// TwinCAT 3 PLC project Untitled1
// ProgramVersion: 3.1.4023.0
// libraries:
//   Tc2_EthernetIP, * (Beckhoff Automation GmbH)
//   Tc2_MC2, * (Beckhoff Automation GmbH)
//   Tc2_Standard, * (Beckhoff Automation GmbH)
//   Tc2_System, * (Beckhoff Automation GmbH)
//   Tc2_TcpIp, * (Beckhoff Automation GmbH)
//   Tc2_Utilities, * (Beckhoff Automation GmbH)
//   Tc3_Interfaces, * (Beckhoff Automation GmbH)
//   Tc3_Module, * (Beckhoff Automation GmbH)
//   VisuDialogs, * (System)
// project tree:
//   DUTs/ ST_Handshake.TcDUT, ST_Input_Output.TcDUT
//   / GlobalTextList.TcGTLO, PlcTask.TcTTO, Visualization Manager.TcVMO (not stored)
//   GVLs/ Global_Variables.TcGVL, GVL.TcGVL
//   POUs/ FB_Server.TcPOU, FB_ServerApplication.TcPOU, FB_ServerConnection.TcPOU, MAIN.TcPOU, Torque.TcPOU, Velocity.TcPOU
//   POUs/Helper POUs/ FB_FrameFifo.TcPOU, FB_LogFifo.TcPOU, F_ADSLOGHEXDATA.TcPOU
//   VISUs/ Visualization.TcVIS
// real-time tasks:
//   TASK PlcTask: cycle T#100us, priority 20, ADS port 350
// motion (NC):
//   TASK NC-Task 1 SAF: cycle T#2ms, priority 4, ADS port 501
//   TASK NC-Task 1 SVB: cycle T#10ms, priority 8, ADS port 511
//   AXIS Axis 1 (id 1)
//     OtherSettings: AllowMotionCmdToSlave=true
//     encoder EncType=4
//       EncPara: MaxCount=#x0000ffff
//         Inc: RefSoftSyncMask=#x0000ffff
//     drive DrvType=24
//       Analog: TorqueSetpointScale=10, ScaleFactorActTorque=0.1
//       TimeComp: TaskDelayCycles=1
//     controller CtrType=1
//       CtrPara: PriorControlFactor=1
//         Observer: BandWidth=20
//   AXIS Axis 2 (id 2)
//     Dynamic: Acceleration=193.102849139388, Deceleration=193.102849139388, Jerk=13.317479191567
//     Velo: RefSearch=28.7326666666667, RefSync=28.7326666666667, SlowManual=143.663333333333, FastManual=861.98, Fast=2873.26666666667, Maximum=2800
//     PositionAreaControl: Enable=false
//     TargetPosControl: Enable=false
//     OtherSettings: AllowMotionCmdToSlave=true
//     encoder EncType=19
//       EncPara: ScaleFactorNumerator=94, ScaleFactorDenominator=1048576, MaxCount=#xffffffff
//     drive DrvType=16
//       DrvPara: MaxCount=#xffffffff
//         Analog: VeloReferenz=3000, VeloScale=32, TorqueSetpointScale=10, ScaleFactorActTorque=0.1
//         TimeComp: TaskDelayCycles=1
//     controller CtrType=1
//       CtrPara: PriorControlFactor=1
//         PosDiffControl: Enable=false
//         Observer: BandWidth=20
//   AXIS Axis 3 (id 3)
//     OtherSettings: AllowMotionCmdToSlave=true
//     encoder EncType=19
//       EncPara: ScaleFactorNumerator=104.8576, ScaleFactorDenominator=1048576, MaxCount=#xffffffff
//     drive DrvType=16
//       DrvPara: MaxCount=#xffffffff, DriveControlDWord=#x00020000
//         Analog: VeloScale=32, TorqueSetpointScale=10, ScaleFactorActTorque=0.1
//         TimeComp: TaskDelayCycles=1
//     controller CtrType=1
//       CtrPara: PriorControlFactor=1
//         Observer: BandWidth=20
// I/O:
//   DEVICE Device 1 (EtherCAT), AmsNetId 192.168.0.4.2.1
//     Term 13 (EK1200) [EK1200-5000 EtherCAT Power supply (2A E-Bus)]
//       Term 14 (EL1004) [EL1004 4Ch. Dig. Input 24V, 3ms]
//       Term 15 (EL1008) [EL1008 8Ch. Dig. Input 24V, 3ms]
//       Term 16 (EL2004) [EL2004 4Ch. Dig. Output 24V, 0.5A]
//       Term 17 (EL2008) [EL2008 8Ch. Dig. Output 24V, 0.5A]
//       Term 18 (EL3102) [EL3102 2Ch. Ana. Input +/-10V, Diff.]
//       Term 19 (EL4132) [EL4132 2Ch. Ana. Output +/-10V, 16bit]
//       Term 20 (EK1110) [EK1110 EtherCAT extension]
//     Term 21 (EK1100) [EK1100 EtherCAT Coupler (2A E-Bus)]
//       Term 22 (EL7031) [EL7031 1Ch. Stepper motor output stage (24V, 1.5A)]
//       Term 23 (EL7211-0010) [EL7211-0010 1Ch. MDP742 Servo motor output stage with OCT (50V, 4.5A RMS)]
//       Term 27 (EL9011) [EL9011 End Terminal]
//     Term 24 (EK1100) [EK1100 EtherCAT Coupler (2A E-Bus)]
//       Term 25 (EL7211-0010) [EL7211-0010 1Ch. MDP742 Servo motor output stage with OCT (50V, 4.5A RMS)]
//       Term 26 (EK1110) [EK1110 EtherCAT extension]
//   DEVICE Device 5 (COM Port)
// variable links:
//   NC-Task 1 SAF/Axes/Axis 2 <-> Device 1 (EtherCAT)/Term 21 (EK1100)/Term 23 (EL7211-0010)
//     Drive/Inputs/In/nDataIn3[0] <-> DRV Torque actual value/Torque actual value
//     Drive/Inputs/In/nDcOutputTime <-> InfoData/DcOutputShift
//     Drive/Inputs/In/nState1 <-> DRV Statusword/Statusword
//     Drive/Inputs/In/nState2 <-> DRV Statusword/Statusword @bit 8
//     Drive/Inputs/In/nState4 @bit 1 <-> WcState/InputToggle
//     Drive/Inputs/In/nState4 <-> WcState/WcState
//     Drive/Outputs/Out/nCtrl1 <-> DRV Controlword/Controlword
//     Drive/Outputs/Out/nCtrl2 <-> DRV Controlword/Controlword @bit 8
//     Enc/Inputs/In/nDataIn1 <-> FB Position/Position
//     Enc/Inputs/In/nDcInputTime <-> InfoData/DcInputShift
//     Enc/Inputs/In/nState4 @bit 1 <-> WcState/InputToggle
//     Enc/Inputs/In/nState4 <-> WcState/WcState
//   NC-Task 1 SAF/Axes/Axis 3 <-> Device 1 (EtherCAT)/Term 24 (EK1100)/Term 25 (EL7211-0010)
//     Drive/Inputs/In/nDcOutputTime <-> InfoData/DcOutputShift
//     Drive/Inputs/In/nState1 <-> DRV Statusword/Statusword
//     Drive/Inputs/In/nState2 <-> DRV Statusword/Statusword @bit 8
//     Drive/Inputs/In/nState4 @bit 1 <-> WcState/InputToggle
//     Drive/Inputs/In/nState4 <-> WcState/WcState
//     Drive/Outputs/Out/nCtrl1 <-> DRV Controlword/Controlword
//     Drive/Outputs/Out/nCtrl2 <-> DRV Controlword/Controlword @bit 8
//     Drive/Outputs/Out/nDataOut2 <-> DRV Target velocity/Target velocity
//     Enc/Inputs/In/nDataIn1 <-> FB Position/Position
//     Enc/Inputs/In/nDcInputTime <-> InfoData/DcInputShift
//     Enc/Inputs/In/nState4 @bit 1 <-> WcState/InputToggle
//     Enc/Inputs/In/nState4 <-> WcState/WcState
//   Untitled1/Untitled1 Instance <-> Device 1 (EtherCAT)/Term 21 (EK1100)/Term 23 (EL7211-0010)
//     PlcTask Outputs/Torque.TorqueLim <-> DRV Torque limitation/Torque limitation
//     PlcTask Outputs/Torque.TorqueVAL <-> DRV Target torque/Target torque
//   Untitled1/Untitled1 Instance <-> NC-Task 1 SAF/Axes/Axis 2
//     PlcTask Inputs/GVL.ActualTorque <-> Outputs/ToPlc/ActTorque
//     PlcTask Inputs/Torque.Axis1.NcToPlc <-> Outputs/ToPlc
//     PlcTask Outputs/Torque.Axis1.PlcToNc <-> Inputs/FromPlc
//   Untitled1/Untitled1 Instance <-> NC-Task 1 SAF/Axes/Axis 3
//     PlcTask Inputs/Velocity.Axis2.NcToPlc <-> Outputs/ToPlc
//     PlcTask Outputs/Velocity.Axis2.PlcToNc <-> Inputs/FromPlc

CONFIGURATION Untitled1
    RESOURCE PLC ON TwinCAT3
        TASK PlcTask(INTERVAL := T#100us, PRIORITY := 20);
        PROGRAM Torque WITH PlcTask : Torque;
        PROGRAM Velocity WITH PlcTask : Velocity;
        PROGRAM MAIN WITH PlcTask : MAIN;
    END_RESOURCE
END_CONFIGURATION

// ---- DUTs/ST_Handshake.TcDUT
TYPE ST_Handshake :
STRUCT
	(* Handshake with Mevea. First package to sent to Mevea. Mevea sends similar, but in diffrent order after connection. These must match.*)
	
	in			: UDINT		:= 3;(* Input parameter amount. 4 byte *)
	out			: UDINT		:= 3;(* Output parameter amount. 4 byte *)
	version	 	: UDINT		:= 1;(* Version. 4 byte *)

	(* Total user data size = 12 byte *)
END_STRUCT
END_TYPE

// ---- DUTs/ST_Input_Output.TcDUT
TYPE ST_Input_Output :
STRUCT
	(* data struct to be transferred with Mevea. Not ideal, but simple to implement and does the trick in this case *)
	
	brake				: LREAL		:= 0;(* 8 byte *)
	rpmin_torqout	 	: LREAL		:= 0;(* 8 byte *)
	rpmout_speedin		: LREAL		:= 0;(* 8 byte *)

	(* Total user data size = 24 bytes *)
END_STRUCT
END_TYPE

// ---- GVLs/Global_Variables.TcGVL
VAR_GLOBAL CONSTANT
	PLCPRJ_BUFFER_SIZE						: UDINT := 1000;	(* Max. internal fifo/receiver buffer size *)
	PLCPRJ_RECEIVE_POLLING_TIME				: TIME := T#0MS;	(* Input polling timer if needed to limit the interval. Not in this case *)
	PLCPRJ_RECEIVE_TIMEOUT					: TIME := T#10S;	(* Timeout when receiving. Start waiting new connection. Usually disconnected by peer error triggers it *)

	(* Some project specific error codes *)
	PLCPRJ_ERROR_RECEIVE_TIMEOUT			: UDINT := 16#8101;(* Receive timeout *)
	PLCPRJ_ERROR_SENDFIFO_OVERFLOW			: UDINT := 16#8102;(* Send fifo overflow *)
	PLCPRJ_ERROR_RECFIFO_OVERFLOW			: UDINT := 16#8103;(* Receive fifo overflow *)
	PLCPRJ_ERROR_INVALID_FRAME_FORMAT		: UDINT := 16#8104;(* Invalid frame format/data *)
	
	PLCPRJ_CRUISE_CONTROL_SET				: LREAL := 20;	(* Max. internal fifo/receiver buffer size *)
END_VAR

// ---- GVLs/GVL.TcGVL
VAR_GLOBAL
	maxSimulationTorque: INT;
	maxSimulationVelocity: INT;
	Actual_Velocity: LREAL;
	ActualTorque AT %I*: LREAL;
	(* Velocity and torque datatype should be given a thought. If there is no reason for int, LREAL would be more suitable *)
	SetVelocity: INT;
	SetTorque: INT;
END_VAR

// ---- POUs/Torque.TcPOU
PROGRAM Torque
VAR
	res1Error: BOOL;
	Step: INT;
	Axis1_MV: MC_MoveVelocity;
	Axis1_Error_Reset: MC_Reset;
	Power1_BufferMode: MC_BufferMode;
	Power1_Override: LREAL;
	Power1_EnableNeg: BOOL;
	Power1_EnablePos: BOOL;
	Power1_Enable: BOOL;
	Axis1_Power: MC_Power;
	Axis1: AXIS_REF;
	Power1_Status: BOOL;
	Power1_Busy: BOOL;
	Power1_error: BOOL;
	Power1_Active: BOOL;
	Power1_ErrorID: UDINT;
	ErrorReset1_Execute: BOOL;
	res1Done: BOOL;
	res1Busy: BOOL;
	res1ErrorID: UDINT;
	MV1_Execute: BOOL;
	MV1_Done: BOOL;
	MV1_Velocity: LREAL;
	MV1_Decceleration: LREAL;
	MV1_Jerk: LREAL;
	MV1_Direction: MC_Direction;
	MV1_Buffermode: MC_BufferMode;
	MV1_InVelocity: BOOL;
	MV1_Busy: BOOL;
	MV1_CommandAborted: BOOL;
	MV1_Error: BOOL;
	MV1_ErrorID: UDINT;
	MV1_Acceleration: LREAL;
	MV1_Accelleration: LREAL;
	MV1_Active: BOOL;
	TorqueVAL AT %Q*: INT;
	TorqueLim AT %Q*: UINT;
	Start1Btn: BOOL;
	PowerOnTorqueBtn: BOOL;
	Stop1Btn: BOOL;
	TorqueEnable: BOOL;
	
	TorqueSim: INT;
END_VAR

//Torque Controlled Servo
	
	//In case of an error with torque controlled servo:
	IF(Power1_error = TRUE OR MV1_Error=TRUE)THEN
		//Step := 10;
	END_IF
	
	//Enables user to set the torque of the servomotor
	IF TorqueEnable  = TRUE THEN
		TorqueVAL := SetTorque;
		TorqueSim := SetTorque*maxSimulationTorque;
	END_IF
	CASE Step OF
		0://Start of the power (in next step), when the PowerOnTorque button will be clicked
			IF (PowerOnTorqueBtn = TRUE) THEN
				Step := 1;
			END_IF
		1://Start the torque control, when the StartTorque button will be clicked
	Axis1_Power(
	Axis:=Axis1,
	Enable := TRUE,
	Enable_Positive := TRUE,
	Enable_Negative := TRUE,
	Override := 100,
	BufferMode := Power1_BufferMode,
	Status => Power1_Status,
	Busy => Power1_Busy,
	Active => Power1_Active,
	Error => Power1_error,
	ErrorID =>Power1_ErrorID);
			IF (Start1Btn = TRUE) THEN
				Step := 2;
				PowerOnTorqueBtn := FALSE;
			END_IF
		2://Stop the motor (in next step), when the StopTorque button will be clicked 
			TorqueLim := 200;
			TorqueEnable := TRUE;
			Start1Btn := FALSE;
			Axis1_MV(
	Axis:= Axis1, 
	Execute:= TRUE, 
	//Velocity:= MV1_Velocity, 
	//Acceleration:= MV1_Accelleration, 
	//Deceleration:= MV1_Decceleration, 
	//Jerk:= MV1_Jerk, 
	//Direction:= MV1_Direction, 
	BufferMode:= MV1_Buffermode, 
	//Options:= MV_Options, 
	InVelocity=> MV1_InVelocity, 
	Busy=> MV1_Busy, 
	Active=> MV1_Active, 
	CommandAborted=> MV1_CommandAborted, 
	Error=> MV1_Error, 
	ErrorID=> MV1_ErrorID);
			IF Stop1Btn = TRUE THEN
				Step:= 3;
				Start1Btn:=FALSE;
			END_IF
		3://Stops motor and gets back to the Power On state
			IF Actual_Velocity = 0 THEN
				Step := 1;
				Stop1Btn:=FALSE;
			END_IF
			MV1_Velocity := 0;
			TorqueEnable := FALSE;
			TorqueVAL := 0;
			
		10://Error Step
			Power1_Enable := FALSE;
			MV1_Execute := FALSE; 
			MV1_Velocity := 0;
			SetTorque := 0;
			TorqueEnable := FALSE;
			ErrorReset1_Execute := TRUE;
			IF res1Done = TRUE THEN
				Step := 0;
			END_IF
			
		END_CASE

	
Axis1_Error_Reset(
	Axis := Axis1,
	Execute := ErrorReset1_Execute,
	Done => res1Done,
	Busy => res1Busy,
	Error => res1Error,
	ErrorID => res1ErrorID);

END_PROGRAM

// ---- POUs/Velocity.TcPOU
PROGRAM Velocity
VAR
	Axis2_Power: MC_Power;
	Axis2: AXIS_REF;
	Power2_EnablePos: BOOL;
	Power2_EnableNeg: BOOL;
	Power2_Enable: BOOL;
	Power2_Override: LREAL;
	Power2_BufferMode: MC_BufferMode;
	Power2_Status: BOOL;
	Power2_Busy: BOOL;
	Power2_Active: BOOL;
	Power2_Error: BOOL;
	Power2_ErrorID: UDINT;
	Axis2_ErrorReset: MC_Reset;
	ErrorReset2_Execute: BOOL;
	res2Done: BOOL;
	res2Busy: BOOL;
	res2Error: BOOL;
	res2ErrorID: UDINT;
	Axis2_MoveVelocity: MC_MoveVelocity;
	MV2_Execute: BOOL;
	MV2_Accelleration: LREAL;
	MV2_Decceleration: LREAL;
	MV2_Jerk: LREAL;
	MV2_Direction: MC_Direction := 1;
	MV2_Buffermode: MC_BufferMode;
	MV2_InVelocity: BOOL;
	MV2_Busy: BOOL;
	MV2_Active: BOOL;
	MV2_CommandAborted: BOOL;
	MV2_Error: BOOL;
	MV2_ErrorID: UDINT;
	StepV: INT;
	PowerOnVelocityBtn: BOOL;
	Start2Btn: BOOL;
	Stop2Btn: BOOL;
	Read_Velocity: MC_ReadActualVelocity;
	RV_Enable: BOOL;
	RV_Valid: BOOL;
	RV_Busy: BOOL;
	RV_Error: BOOL;
	RV_ErrorID: UDINT;
	A_Velocity: LREAL;
	MV2_Velocity: LREAL;
	RES_BUTTON: BOOL;
	errorDiode: BOOL;
	VelocitySim: INT;
END_VAR

//Axis2 - Velocity controlled servomotor
//Velocity Controlled Servo
		VelocitySim:=maxSimulationVelocity*ActualVelocity/2000;
		IF (SetVelocity<0)THEN
			MV2_Direction := MC_Positive_Direction;
		ELSE
			MV2_Direction := MC_Negative_Direction;
		
		END_IF
		//In case of an error with torque controlled servo:
	IF(Power2_error = TRUE OR MV2_Error=TRUE) THEN
		//StepV := 10;
		//Servomotor was stopped with external force
		IF	MV2_ErrorID=17744 THEN
			StepV := 11;
			errorDiode :=TRUE;
		END_IF
	END_IF
		
		CASE StepV OF
		0://Start of the power (in next step), when the PowerOnVelocity button will be clicked
			IF (PowerOnVelocityBtn = TRUE) THEN
				StepV := 1;
			END_IF
		1://Start the torque control, when the StartTorque button will be clicked
			Axis2_Power(
	Axis:= Axis2, 
	Enable:= TRUE, 
	Enable_Positive:= TRUE, 
	Enable_Negative:= TRUE, 
	Override:= 100, 
	BufferMode:= Power2_BufferMode, 
	//Options:= , 
	Status=> Power2_Status, 
	Busy=> Power2_Busy, 
	Active=> Power2_Active, 
	Error=> Power2_Error, 
	ErrorID=> Power2_ErrorID);
	RV_Enable:=TRUE;
			IF (Start2Btn = TRUE) THEN
				StepV := 2;
				PowerOnVelocityBtn :=FALSE;
			END_IF
		2://Stop the motor (in next step), when the StopVelocity button will be clicked
			Axis2_MoveVelocity(
	Axis:= Axis2, 
	Execute:=TRUE, 
	Velocity:= MV2_Velocity, 
	Acceleration:= 2000, 
	Deceleration:= 2000, 
	Jerk:= 20000, 
	Direction:= MV2_Direction, 
	BufferMode:= MV2_Buffermode, 
	//Options:= MV_Options, 
	InVelocity=> MV2_InVelocity, 
	Busy=> MV2_Busy, 
	Active=> MV2_Active, 
	CommandAborted=> MV2_CommandAborted, 
	Error=> MV2_Error, 
	ErrorID=> MV2_ErrorID);
			IF NOT(MV2_Velocity = SetVelocity) THEN
				IF(SetVelocity>0)THEN
					MV2_Velocity := SetVelocity;
				ELSE
						MV2_Velocity := -SetVelocity;
				END_IF
				MV2_Execute := FALSE; 
			END_IF
			IF Stop2Btn = TRUE THEN
				StepV:= 3;
				Start2Btn:=FALSE;
			END_IF
		3://Stops motor and gets back to the Power On state
			IF Actual_Velocity <= 0 THEN
				MV2_Execute := TRUE;
				StepV := 1;
				Stop2Btn := FALSE;
			END_IF
			MV2_Execute := FALSE;
			MV2_Velocity := 0;
			
						
			
		10://Error Step
			Power2_Enable := FALSE;
			MV2_Execute := FALSE; 
			MV2_Velocity := 0;
			ErrorReset2_Execute := TRUE;
			IF res2Done = TRUE THEN
				StepV := 0;
			END_IF
			
			11:
			Stop2Btn:=FALSE;
			Start2Btn:=FALSE;
			PowerOnVelocityBtn:=FALSE;
			IF(RES_BUTTON)THEN
			MV2_Execute:=FALSE;
			Axis2_Power(
				Axis:= Axis2, 
				Enable:= FALSE);
			ErrorReset2_Execute:=TRUE;
			IF(res2Done)THEN
				ErrorReset2_Execute:=FALSE;
				errorDiode := FALSE;
				StepV :=0;
			END_IF
			END_IF
			
			
		END_CASE


	
	Axis2_ErrorReset(
	Axis := Axis2,
	Execute := ErrorReset2_Execute,
	Done => res2Done,
	Busy => res2Busy,
	Error => res2Error,
	ErrorID => res2ErrorID);
	
	Axis2_MoveVelocity(
	Axis:= Axis2, 
	Execute:=MV2_Execute, 
	//Options:= MV_Options, 
	InVelocity=> MV2_InVelocity, 
	Busy=> MV2_Busy, 
	Active=> MV2_Active, 
	CommandAborted=> MV2_CommandAborted, 
	Error=> MV2_Error, 
	ErrorID=> MV2_ErrorID);
	
	Read_Velocity(
	Axis:= Axis2, 
	Enable:= RV_Enable, 
	Valid=> RV_Valid, 
	Busy=> RV_Busy, 
	Error=> RV_Error, 
	ErrorID=> RV_ErrorID, 
	ActualVelocity=> A_Velocity);
	Actual_Velocity:=-A_Velocity;

END_PROGRAM

// ---- POUs/MAIN.TcPOU
PROGRAM MAIN
VAR
	//sSrvNetID		: T_AmsNetID	:= '193.167.148.78.1.1';(* TwinCAT TCP/IP server network address *)
	//sLocalHost		: T_Ipv4Addr 	:= '192.168.0.5';(* Server IP network address *)
	//nLocalPort		: UDINT 		:= 5111;(* Server port number *)
	sSrvNetID		: T_AmsNetID	:= '';(* TwinCAT TCP/IP server network address *)
	sLocalHost		: T_Ipv4Addr 	:= '127.0.0.1';(* Server IP network address *)
	nLocalPort		: UDINT 		:= 5111;(* Server port number *)
	bEnable			: BOOL 			:= TRUE;(* TRUE => Enable server data exchange, FALSE => Disable *)
	bLog			: BOOL			:= FALSE;(* TRUE => Enable log message output, FALSE => Disable *)
	fbServer		: FB_Server := ( sPrefix := 'SERVER::' );(* Server (connection) instance *)
	hServer			: T_HSERVER;(* Server connection handle *)

	fbCloseAll		: FB_SocketCloseAll;
	bInitialize		: BOOL := TRUE;
END_VAR

(* Before running this install TF6310 library from Beckhoff infosys to PC or PLC respectively *)

(* On PLC reset or program download close all old (opened) connections *)
fbCloseAll( sSrvNetID := sSrvNetID, bExecute:= bInitialize );
IF fbCloseAll.bBusy OR fbCloseAll.bError THEN
	RETURN;
END_IF

IF bInitialize THEN
	bInitialize := FALSE;

	(* Initialize server handle *)
	F_CreateServerHnd( 	sSrvNetID 	:= sSrvNetID,
						sLocalHost 	:= sLocalHost,
						nLocalPort	:= nLocalPort,
						nMode 		:= SEL( bLog, 0, CONNECT_MODE_ENABLEDBG ),(* Enable debug messages *)
						bEnable 	:= FALSE,(* TRUE = leave listener socket open, FALSE = close listener socket after last connection ist closed too *)
						hServer 	:= hServer );
END_IF


(* Trigger the execution of every server (connection) instance *)
fbServer( hServer := hServer, sSrvNetID := sSrvNetID, bEnable := bEnable, bLog := bLog );

END_PROGRAM

// ---- POUs/FB_Server.TcPOU
FUNCTION_BLOCK FB_Server
VAR_IN_OUT
	hServer			: T_HSERVER;(* Server connection handle *)
END_VAR
VAR_INPUT
	sSrvNetID		: T_AmsNetID	:= '';(* TwinCAT TCP/IP server network address *)
	bEnable			: BOOL 			:= FALSE;(* TRUE => Enable server data exchange, FALSE => Disable *)
	bLog			: BOOL 			:= FALSE;(* TRUE => Enable log message output, FALSE => Disable *)
	sPrefix			: STRING 		:= 'SERVER::';(* Log message description string (allows the identification of log message source) *)
END_VAR
VAR_OUTPUT
	eState			: E_SocketConnectionState := eSOCKET_DISCONNECTED;(* TCP/IP connection state *)
END_VAR
VAR
	fbApplication 	: FB_ServerApplication;(* Server application control function block *)
	fbConnection	: FB_ServerConnection;(* Server data exchange control function block *)
	fbTx 			: FB_FrameFifo;(* Tx fifo *)
	fbRx 			: FB_FrameFifo;(* Rx fifo *)
	fbLog			: FB_LogFifo;(* Log/debug/error fifo *)
END_VAR

(*-------------------------- Trigger data exchange -----------------------------------------------*)
fbConnection( 	hServer := hServer, sSrvNetID := sSrvNetID, 
				fbRx := fbRx, fbTx := fbTx, fbLog := fbLog, 
				bEnable := bEnable, bLog := bLog, sPrefix := sPrefix, eState=>eState );
	
IF fbConnection.eState = eSOCKET_CONNECTED THEN(* Connection established *)
	fbApplication( fbTx := fbTx, fbRx := fbRx, fbLog := fbLog );
END_IF

END_FUNCTION_BLOCK

// ---- POUs/FB_ServerApplication.TcPOU
(* Sample server application. Adapt this code to match your needs. *)
FUNCTION_BLOCK FB_ServerApplication
VAR_IN_OUT
	fbTx 			: FB_FrameFifo;(* TX fifo *)
	fbRx 			: FB_FrameFifo;(* RX fifo *)
	fbLog			: FB_LogFifo;(* Log message fifo *)
END_VAR
VAR
	stToClient		: ST_Input_Output; (* Tx user data *)
	stFromClient	: ST_Input_Output; (* Rx user data *)
	sLogMessage 	: T_MaxString := '';(* Log/debug/error message *)
	velInputControl	: LREAL := 0;
	torqPidControl: FB_BasicPID;
	resetPID		: BOOL := TRUE;
	PIDval			: LREAL := 0;
END_VAR

(*------------------- Fetch rx data and send them back to the client -------------------------------------------------- *)
REPEAT
	fbRx.RemoveHead( );(* Fetch data from rx fifo *)
	IF fbRx.bOk THEN(* Success *)
		stFromClient := fbRx.stGet;
		velInputControl := stFromClient.rpmout_speedin;
		
		(* Following PID controller is the crise control. This emulates the intelligent machine throttle/brake. *)
		(* ToDo find some reasonable PID parameters *)
		torqPidControl(
			fSetpointValue:= PLCPRJ_CRUISE_CONTROL_SET, 
			fActualValue:= velInputControl, 
			bReset:= resetPID, 
			fCtrlCycleTime:= 0.00025, 
			fKp:= 120,
			fTn:= 2, 
			fTv:= 1, 
			fTd:= 0.2);
		IF torqPidControl.fCtrlOutput >= 600 THEN
			PIDval := 600;
		ELSIF torqPidControl.fCtrlOutput <= -600 THEN
			PIDval := -600;
		ELSE
			PIDval := torqPidControl.fCtrlOutput;
		END_IF
		resetPID := FALSE;
		(* Set the got and calculated values. First to servos and then to Mevea *)
		(* Velocity is the angular velocity of the motor. Should be scaled possibly *)
		SetVelocity :=REAL_TO_INT(velInputControl);
		(* Max torque is set to +-600. Can be adjusted from mevea *)
		SetTorque := REAL_TO_INT(PIDval);
		
		stToClient.brake :=0;
		stToClient.rpmin_torqout :=PIDval;
		stToClient.rpmout_speedin :=1;

		(* Send data back to the client *)
		fbTx.AddTail( stPut := stToClient );(* Put user data to the tx fifo *)
		IF NOT fbTx.bOk THEN(* Fifo overflow => Log error *)
			fbLog.Error( sMessage := 'FB_FrameFifo(sender)', nErrID := PLCPRJ_ERROR_SENDFIFO_OVERFLOW );
		END_IF
	END_IF
UNTIL NOT fbRx.bOk
END_REPEAT

(*---------------------- Get log/error messages from log fifo ------------------*)
REPEAT
	fbLog.Remove( );
	IF fbLog.bOk THEN

		(* TODO: Implement log message handler *)
		sLogMessage := fbLog.sGet;

	END_IF
UNTIL NOT fbLog.bOk
END_REPEAT

END_FUNCTION_BLOCK

// ---- POUs/Helper POUs/FB_FrameFifo.TcPOU
(* Tx/Rx (string data) fifo control function block *)
FUNCTION_BLOCK FB_FrameFifo
VAR_INPUT
	bLog		: BOOL		:= FALSE;(* TRUE => Enable log message output, FALSE => Disable *)
	sPrefix		: STRING	:= 'Unknown::';(* Log message description string (allows the identification of log message source) *)
	stPut		: ST_Input_Output;(* Frame to add (write) to the fifo *)
END_VAR
VAR_OUTPUT
	bOk			: BOOL; 	(* TRUE = New entry added or removed succesfully, FALSE = Fifo overflow or fifo empty *)
	stGet		: ST_Input_Output;(* Frame removed (read) from fifo *)
	nCount		: UDINT		:= 0;(* Number of fifo entries *)
	cbFree		: UDINT 	:= 0;(* Free buffer space *)
END_VAR
VAR
	fbBuffer 	: FB_MemRingBuffer;(* Basic (lower level) buffer control function block *)
	buffer		: ARRAY[-3..PLCPRJ_BUFFER_SIZE] OF BYTE;(* Internal buffer memory *)
END_VAR

;

ACTION AddTail:
(* Adds new fifo entry *)
fbBuffer.A_AddTail( pBuffer:= ADR(buffer), cbBuffer:= SIZEOF(buffer),
					pWrite := ADR( stPut ), cbWrite := SIZEOF( stPut ), 
					bOk=>bOk, nCount=>nCount );
IF bOk THEN
	cbFree := PLCPRJ_BUFFER_SIZE - fbBuffer.cbSize;(* Calculate the free buffer space *)
	IF bLog THEN(* Log message *)
		F_ADSLOGHEXDATA( CONCAT( sPrefix, '<=' ), ADR( stPut ), SIZEOF( stPut ) );
	END_IF
END_IF
END_ACTION

ACTION Clear:
(* Resets fifo = clears all data *)
MEMSET( ADR( stGet ), 0, SIZEOF( stGet ) );
fbBuffer.A_Reset( pBuffer:= ADR(buffer), cbBuffer:= SIZEOF(buffer),
					pWrite := ADR( stPut ), cbWrite := SIZEOF( stPut ), 
					pRead := ADR( stGet ), cbRead := SIZEOF( stPut ),
					bOk=>bOk, nCount=>nCount );
cbFree := PLCPRJ_BUFFER_SIZE;(* Free buffer size *)
END_ACTION

ACTION RemoveHead:
(* Removes oldest fifo entry *)
MEMSET( ADR( stGet ), 0, SIZEOF( stGet ) );
fbBuffer.A_RemoveHead( pBuffer:= ADR(buffer), cbBuffer:= SIZEOF(buffer),
						pRead := ADR( stGet ), cbRead := SIZEOF( stGet ),
						bOk=>bOk, nCount=>nCount );
IF bOk THEN
	cbFree := PLCPRJ_BUFFER_SIZE - fbBuffer.cbSize;(* Calculate the free buffer space *)
END_IF
END_ACTION

END_FUNCTION_BLOCK

// ---- POUs/Helper POUs/F_ADSLOGHEXDATA.TcPOU
(* This function logs hexadecimal data to the TwinCAT XAE->Error list window *)
FUNCTION F_ADSLOGHEXDATA : DINT
VAR_INPUT
	sPrefix		: STRING;(* Debug message prefix string (allows the identification of log message source) *)
	pBuffer		: PVOID;(* Address of source buffer *)
	cbBuffer	: UDINT;(* Byte size of source buffer *)
END_VAR
VAR
	fbSplit	: FB_MemBufferSplit;
	sArg	: T_MaxString;
	sFormat : STRING;
END_VAR

IF pBuffer = 0 OR cbBuffer = 0 THEN
	RETURN;
END_IF

sFormat := CONCAT( sPrefix, '%s' );
fbSplit.eCmd := eEnumCmd_First;

REPEAT
	fbSplit( pBuffer := pBuffer, cbBuffer := cbBuffer, cbSize := 32 );(* Split binary data to 32 byte segments *)
	IF fbSplit.bOk THEN

		sArg := DATA_TO_HEXSTR( pData := fbSplit.pSegment, cbData := fbSplit.cbSegment, FALSE );(* Convert binary data to hex string *)

		F_ADSLOGHEXDATA := ADSLOGSTR( ADSLOG_MSGTYPE_HINT OR ADSLOG_MSGTYPE_LOG, sFormat, sArg );(* Log hex string *)

		sFormat := '%s';
		fbSplit.eCmd := eEnumCmd_Next;
	END_IF
UNTIL NOT fbSplit.bOk
END_REPEAT

END_FUNCTION

// ---- POUs/Helper POUs/FB_LogFifo.TcPOU
(* Log/debug/error message fifo *)
FUNCTION_BLOCK FB_LogFifo
VAR_INPUT
	bLog		: BOOL 		:= FALSE;(* TRUE => Enable log message output, FALSE => Disable *)
	sPrefix		: STRING 	:= 'Unknown::';(* Log message description string (allows the identification of log message source) *)
	
	sMessage	: STRING 	:= '';(* String message to add (write) to the fifo *)
	nErrID		: UDINT 	:= 0;(* Error code to add (write) to the fifo *)
	hSocket		: T_HSOCKET;(* Socket connection handle *)
END_VAR
VAR_OUTPUT
	bOk			: BOOL;(* TRUE = New entry added or removed succesfully, FALSE = Fifo overflow or fifo empty *)
	sGet		: T_MaxString := '';(* String entry removed (read) from fifo *)
	nCount		: UDINT := 0;(* Number of fifo entries *)
END_VAR
VAR
	fbBuffer 	: FB_StringRingBuffer;(* Basic (lower level) string buffer control function block *)
	buffer		: ARRAY[0..PLCPRJ_BUFFER_SIZE] OF BYTE;(* Internal buffer memory *)
	sSource		: T_MaxString;	
	sPut		: T_MaxString;
END_VAR

;

ACTION Clear:
(* Clears all fifo entries *)
fbBuffer.A_Reset( 	pBuffer := ADR( buffer ), cbBuffer := SIZEOF( buffer ), 
					bOk=>bOk, nCount=>nCount, getValue=>sGet );
END_ACTION

ACTION Error:
(* Adds new fifo entry *)
IF nErrID = 0 THEN
	sSource := '::Error: 0x';
ELSIF ( nErrID AND 16#80000000) = 16#80000000 THEN
	IF nErrID = 16#80072746 THEN
		sSource := '::Win32 error (the connection is reset by remote side): 0x';
	ELSE
		sSource := '::Win32 error: 0x';
	END_IF
ELSIF (nErrID AND 16#00008100) = 16#00008100 THEN
	CASE nErrID OF
		PLCPRJ_ERROR_RECEIVE_TIMEOUT:
			sSource := '::PLC sample project receive timeout error: 0x';
		PLCPRJ_ERROR_SENDFIFO_OVERFLOW:
			sSource := '::PLC sample project send fifo overflow error: 0x';
		PLCPRJ_ERROR_RECFIFO_OVERFLOW:
			sSource := '::PLC sample project receive fifo overflow error: 0x';
		PLCPRJ_ERROR_INVALID_FRAME_FORMAT:
			sSource := '::PLC sample project invalid frame format error: 0x';
	ELSE
		sSource := '::Other PLC sample project error: 0x';
	END_CASE
ELSIF (nErrID AND 16#00008000) = 16#00008000 THEN
	sSource := '::Internal TCP/IP Connection Server error: 0x';
ELSE
	sSource := '::TwinCAT System error: 0x';
END_IF

sPut := CONCAT( CONCAT( CONCAT( sPrefix, sMessage ), sSource ), DWORD_TO_HEXSTR( nErrID AND 16#FFFF, 0, FALSE ) ); 

fbBuffer.A_AddTail( pBuffer:= ADR(buffer), cbBuffer:= SIZEOF(buffer),
					putValue:= sPut, bOk=>bOk, nCount=>nCount );
IF bOk THEN
	IF bLog THEN(* Log error message *)
		ADSLOGSTR( ADSLOG_MSGTYPE_ERROR OR ADSLOG_MSGTYPE_LOG, '%s', sPut );	
	END_IF
END_IF
END_ACTION

ACTION Message:
(* Adds new fifo entry *)
sPut := CONCAT( CONCAT( sPrefix, sMessage ), CONCAT( '::', HSOCKET_TO_STRING(hSocket) ) );
fbBuffer.A_AddTail( pBuffer:= ADR(buffer), cbBuffer:= SIZEOF(buffer),
					putValue:= sPut, bOk=>bOk, nCount=>nCount );
IF bOk THEN
	IF bLog THEN(* Log information message *)
		ADSLOGSTR( ADSLOG_MSGTYPE_HINT OR ADSLOG_MSGTYPE_LOG, '%s', sPut );	
	END_IF
END_IF
END_ACTION

ACTION Remove:
(* Removes oldest fifo entry *)
IF nCount = 0 THEN
	sGet := '';
	bOk := FALSE;
	RETURN;
END_IF

fbBuffer.A_RemoveHead( pBuffer:= ADR(buffer), cbBuffer:= SIZEOF(buffer),
						getValue=>sGet, bOk=>bOk, nCount=>nCount );
END_ACTION

END_FUNCTION_BLOCK

// ---- POUs/FB_ServerConnection.TcPOU
(* 	This function block implements simple TCP/IP server protocol. *)
FUNCTION_BLOCK FB_ServerConnection
VAR_IN_OUT
	hServer		: T_HSERVER;(* Server connection handle *)
	fbTx 		: FB_FrameFifo;(* TX fifo *)
	fbRx 		: FB_FrameFifo;(* RX fifo *)
	fbLog		: FB_LogFifo;(* Log message fifo *)
END_VAR
VAR_INPUT
	sSrvNetID	: T_AmsNetID	:= '';(* TwinCAT TCP/IP server network address *)
	bEnable		: BOOL			:= FALSE;(* TRUE => Enable/connect, FALSE => Disable/disconnect *)
	tReconnect	: TIME 			:= T#1S;(* Try to reconnect after this time *)
	bLog		: BOOL 			:= FALSE; (* TRUE => Enable debug output, FALSE => Disable debug output *)
	sPrefix		: STRING 		:= 'SERVER::';(* Log message description string (allows the identification of log message source) *)
END_VAR
VAR_OUTPUT
	eState		: E_SocketConnectionState := eSOCKET_DISCONNECTED;(* TCP/IP connection state *)
END_VAR
VAR
	fbConnect 	: FB_ServerClientConnection;(* Create/release TCP/IP connection *)
	fbSend		: FB_SocketSend;(* Send TCP/IP data *)
	fbReceive	: FB_SocketReceive;(* Receive TCP/IP data *)
	nState 		: BYTE;(* Global state *)
	bSndBusy 	: BOOL;(* Tx state *)
	bRcvBusy 	: BOOL;(* Rx state *)
	bDisconnect	: BOOL;(* Disconnect flag, if set the socket will be closed *)

	fbPollTimer	: TON;(* Rx data poll timer *)
	fbRequestTimer	: TON;(* Request timeout timer *)
	fbReconnectTimer : TON;(* Reconnect timer *)

	nS			: UDINT;(* Send frame counter *)
	nR			: UDINT;(* Received frame counter *)
	cbReceived	: UDINT;(* Count of received data bytes *)
	rxBuffer	: ARRAY[0..PLCPRJ_BUFFER_SIZE] OF BYTE;
	cbFrame		: UDINT;(* Rx frame byte size *)
	stTxFrame	: ST_Input_Output;(* Tx frame buffer*)
	stRxFrame	: ST_Input_Output;(* Rx frame buffer*)
	stHandshakeFrame	: ST_Handshake;(* Rx frame buffer (inclusive header) *)
	bAbort		: BOOL;(* Flag to abort frame parsing loop *)
	handshake	: BOOL :=TRUE;
END_VAR

CASE nState OF
	0:(* Create TCP/IP connection *)
		fbConnect( 	eMode := eACCEPT_ALL, tReconnect := tReconnect, bEnable := bEnable, 
					hServer := hServer, eState => eState );
		IF NOT fbConnect.bBusy THEN
			IF NOT fbConnect.bError THEN
				IF eState = eSOCKET_CONNECTED THEN(* we are connected *)
					
					fbTx.Clear( sPrefix := CONCAT( sPrefix, 'FB_FrameFifo(sender)::' ), bLog := bLog );(* Clear TX fifo (optional) *)
					fbRx.Clear( sPrefix := CONCAT( sPrefix, 'FB_FrameFifo(receiver)::' ), bLog := bLog );(* Clear RX fifo (optional) *)
					fbLog.Clear( sPrefix := sPrefix, bLog := bLog );(* Clear log fifo (optional) *)
					bSndBusy := FALSE;
					bRcvBusy := FALSE;
					bDisconnect := FALSE;
					cbReceived 	:= 0;(* Reset number of received data bytes *)
					nR 			:= 0;(* Reset receive frame counter *)
					nS 			:= 0;(* Reset send frame counter *)

					fbPollTimer( IN := FALSE, PT := T#0S );
					fbRequestTimer( IN := FALSE, PT := PLCPRJ_RECEIVE_TIMEOUT );
					fbReconnectTimer( IN := FALSE, PT := tReconnect );
				
					fbLog.Message( sMessage := 'Connection established!', hSocket := fbConnect.hSocket );
					nState 	:= 1;
				END_IF
			ELSE(* Connect error => log error *)
				fbLog.Error( sMessage := 'FB_ServerClientConnection()', nErrID := fbConnect.nErrId );
			END_IF
		END_IF


	1:(* Data exchange state *)
		bDisconnect := NOT bEnable OR bDisconnect;(* User/internal disconnect requested? *)
		IF bDisconnect AND NOT bSndBusy AND NOT bRcvBusy THEN
			bDisconnect := FALSE;
			fbLog.Message( sMessage := 'Closing connection!', hSocket := fbConnect.hSocket );
			nState := 2;(* Disconnect *)
		ELSE

			(* ----------------------- Get/fetch rx data -------------------------------- *)
			IF NOT bDisconnect AND NOT bRcvBusy THEN
				fbPollTimer( IN := TRUE );
				IF fbPollTimer.Q THEN
					IF fbRx.cbFree >= SIZEOF(stRxFrame) THEN(* Check free rx fifo space *)
						fbPollTimer( IN := FALSE, PT := PLCPRJ_RECEIVE_POLLING_TIME );
						fbReceive( bExecute := FALSE );
						fbReceive( 	sSrvNetId	:= sSrvNetID,
									hSocket		:= fbConnect.hSocket,
									cbLen		:= SIZEOF(rxBuffer) - cbReceived,
									pDest		:= ADR(rxBuffer) + cbReceived,
									bExecute	:= TRUE );
						bRcvBusy := TRUE;
					END_IF
				END_IF
				
			ELSE(* Wait until receive not busy *)
				
				fbReceive( bExecute := FALSE );
				IF NOT fbReceive.bBusy THEN
					bRcvBusy := FALSE;
					IF NOT fbReceive.bError THEN
						IF fbReceive.nRecBytes > 0 THEN (* Some bytes received *)

							fbPollTimer( IN := FALSE, PT := T#0S );(* Bytes received => increase the read (polling) speed *)
							fbRequestTimer( IN := FALSE );(* Bytes received => disable timeout check *)
							cbReceived := cbReceived + fbReceive.nRecBytes;

							(* Parse received bytes *)
							REPEAT
								bAbort := TRUE;(* Set flag *)
								
								IF cbReceived >= SIZEOF(stRxFrame) AND NOT handshake THEN (* All header bytes received => check header data *)
									
									MEMCPY( ADR( stRxFrame ), ADR( rxBuffer ), SIZEOF( stRxFrame ) );(* Get header data *)
									
										cbFrame := SIZEOF(stRxFrame);(* Calculate the expected receive frame length *)
										IF cbReceived >= cbFrame  THEN (* All frame (user data) bytes received? *)
	
											MEMCPY( ADR( stRxFrame ), ADR( rxBuffer ), MIN( SIZEOF(stRxFrame), cbFrame ) );
											fbRx.AddTail( stPut := stRxFrame );(* Add user data to the rx fifo *)
											IF fbRx.bOk THEN
												nR := nR + 1;(* Increment receive counter *)

												MEMMOVE( ADR( rxBuffer ), ADR( rxBuffer ) + cbFrame, cbReceived - cbFrame );(* Shift the remaining rx bytes *)
												cbReceived := cbReceived - cbFrame;(* Recalculate the size of the remaining rx bytes *)

												IF fbRx.cbFree >= SIZEOF(stRxFrame) THEN
													bAbort := FALSE;(* reset flag, try to parse next frame *)
												END_IF
											ELSE (* Fifo overflow => log error and disconnect *)
												fbLog.Error( sMessage := 'FB_FrameFifo(receiver)', nErrID := PLCPRJ_ERROR_RECFIFO_OVERFLOW );
												bDisconnect := TRUE;(* Set flag *)
												RETURN;
											END_IF

(*										ELSE repeat reading *)
										END_IF
								ELSIF cbReceived >= SIZEOF(stHandshakeFrame) AND handshake THEN
									handshake := FALSE;
									cbFrame := SIZEOF(stHandshakeFrame);
									MEMCPY( ADR( stHandshakeFrame ), ADR( rxBuffer ), cbFrame );
									fbSend(	sSrvNetID 	:= sSrvNetID,
										hSocket		:= fbConnect.hSocket,
										cbLen		:= SIZEOF(stHandshakeFrame),(* Size of header + size of user data *)
										pSrc		:= ADR(stHandshakeFrame),(* Pointer to the frame data *)
										bExecute	:= TRUE );
									MEMMOVE( ADR( rxBuffer ), ADR( rxBuffer ) + cbFrame, cbReceived - cbFrame );(* Shift the remaining rx bytes *)
									cbReceived := cbReceived - cbFrame;(* Recalculate the size of the remaining rx bytes *)

(*								ELSE repeat reading *)
								END_IF (* IF cbReceived >= SIZEOF(stRxFrame.head) THEN *)

							UNTIL bAbort
							END_REPEAT

						ELSE(* No bytes received *)
							fbRequestTimer( IN := TRUE );(* No bytes received => enable timeout check *)
							IF fbRequestTimer.Q THEN (* Timeout error*)
								fbRequestTimer( IN := FALSE );
								fbLog.Error( sMessage := 'FB_ServerConnection()', nErrID := PLCPRJ_ERROR_RECEIVE_TIMEOUT );
								bDisconnect := TRUE;(* Set flag *)
							END_IF							
						END_IF(* IF fbReceive.nRecBytes > 0 THEN *)

					ELSE(* Receive error => Log error and disconnect *)
						fbLog.Error( sMessage := 'FB_SocketReceive()', nErrID := fbReceive.nErrId );
						bDisconnect := TRUE;(* set flag *)
					END_IF

				END_IF(* IF NOT fbReceive.bBusy THEN *)
				
			END_IF(* IF NOT bDisconnect AND NOT bRcvBusy THEN *)
			(* -------------------------------------------------------------------------- *)

			
			
			(* ------------------------------ Send tx data ------------------------------ *)
			IF NOT bDisconnect AND NOT bSndBusy THEN
				fbTx.RemoveHead();(* Remove oldest user data entry *)
				IF fbTx.bOk THEN(* Success *)
						
					stTxFrame := fbTx.stGet;
					
					(* Send frame *)
					fbSend( bExecute := FALSE );
					fbSend(	sSrvNetID 	:= sSrvNetID,
							hSocket		:= fbConnect.hSocket,
							cbLen		:= SIZEOF(stTxFrame),(* Size of header + size of user data *)
							pSrc		:= ADR(stTxFrame),(* Pointer to the frame data *)
							bExecute	:= TRUE );
					bSndBusy := TRUE;
				END_IF
			ELSE(* Wait until send not busy *)
				fbSend( bExecute := FALSE );
				IF NOT fbSend.bBusy THEN
					bSndBusy := FALSE;
					IF NOT fbSend.bError THEN(* No error *)
						nS := nS + 1;(* Increment the number of send frames *)
					ELSE(* Send error => Log error and disconnect *)
						fbLog.Error( sMessage := 'FB_SocketSend()', nErrID := fbSend.nErrId );
						bDisconnect := TRUE;(* Set flag *)
					END_IF
				END_IF
			END_IF
			(* -------------------------------------------------------------------------- *)

			
		END_IF(* IF bDisconnect AND NOT bSndBusy AND NOT bRcvBusy THEN *)


	2:(* Disconnect *)
		fbConnect( hServer := hServer, bEnable:= FALSE, eState=>eState );
		IF eState = eSOCKET_DISCONNECTED THEN
			handshake := TRUE;
			fbReconnectTimer( IN := TRUE );(* Please wait some seconds and then try to connect again *)
			IF fbReconnectTimer.Q THEN
				fbReconnectTimer( IN := FALSE );
				nState := 0;
			END_IF
		END_IF

END_CASE

END_FUNCTION_BLOCK

// ---- GlobalTextList.TcGTLO
TEXTLIST GlobalTextList
  262 = '0'
  411 = '1'
  447 = '10'
  924 = 'Actual Torque'
  13 = 'Actual Velocity'
  391 = 'Error caused by external force'
  680 = 'GroupBox'
  550 = 'Label'
  38 = 'Power On'
  956 = 'Power On Torque'
  697 = 'Power On Velocity'
  351 = 'RESET'
  703 = 'Set te torque:'
  56 = 'Set the torque:'
  290 = 'Simualted Velocity:'
  637 = 'Simulated Torque'
  84 = 'Start'
  327 = 'Start Torque'
  923 = 'Start Velocity'
  707 = 'Stop'
  904 = 'Stop Torque'
  901 = 'Stop Velocity'
  848 = 'Torque'
  141 = 'Velocity'
  392 = 'Velocity:'
END_TEXTLIST

// ---- VISUs/Visualization.TcVIS
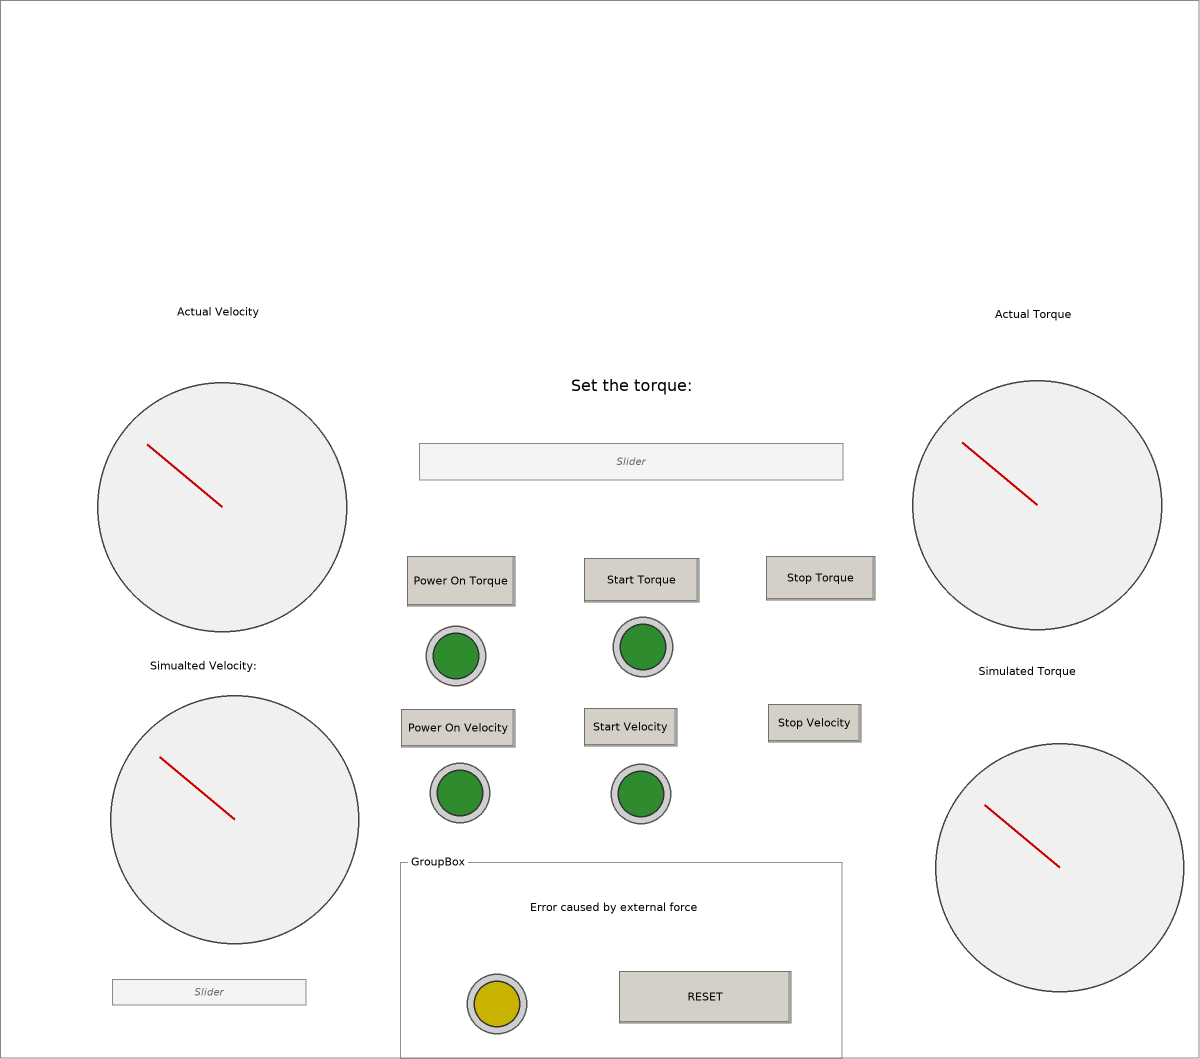
VISUALIZATION Visualization  // 1200x1059
    Slider (419,443 424x37), variable: SetTorque, scale -150..150
    Button (584,558 115x44), "Start Torque"
        OnMouseClick: toggle Torque.Start1Btn
    Button (407,556 108x50), "Power On Torque"
        OnMouseClick: toggle Torque.PowerOnTorqueBtn
    Button (766,556 109x44), "Stop Torque"
        OnMouseClick: toggle Torque.Stop1Btn
    Label (532,358 200x55), "Set the torque:"
    Button (401,709 114x38), "Power On Velocity"
        OnMouseClick: toggle Velocity.PowerOnVelocityBtn
    Button (584,708 93x38), "Start Velocity"
        OnMouseClick: toggle Velocity.Start2Btn
    Button (768,704 93x38), "Stop Velocity"
        OnMouseClick: toggle Velocity.Stop2Btn
    Meter360 (97,382 250x250), value: Actual_Velocity, style: Meter-Meter360-Gray, scale format: %.1f, scale 0..2000
    Label (141,646 125x40), "Simualted Velocity:"
    Meter360 (912,380 250x250), value: ActualTorque, style: Meter-Meter360-Gray, scale format: %.1f, scale -12..12
    Lamp1 (421,621 70x70), variable: Torque.Power1_Active, style: Lamp-Lamp1-Green
    Lamp1 (608,612 70x70), variable: Torque.TorqueEnable, style: Lamp-Lamp1-Green
    Lamp1 (606,759 70x70), variable: Velocity.Start2Btn, style: Lamp-Lamp1-Green
    Lamp1 (425,758 70x70), variable: Velocity.Power2_Active, style: Lamp-Lamp1-Green
    Slider (112,979 194x26), variable: SetVelocity, scale 0..1000
    Label (96,267 244x90), "Actual Velocity"
    Label (888,270 291x89), "Actual Torque"
    Meter360 (94,695 281x249), value: Velocity.VelocitySim, style: Meter-Meter360-Gray, scale format: %.1f, scale 0..100
    Meter360 (919,743 281x249), value: Torque.TorqueSim, style: Meter-Meter360-Gray, scale format: %.1f, scale 0..100
    Label (882,627 291x89), "Simulated Torque"
    GroupBox (400,854 442x205), "GroupBox"
        Button (219,117 172x52), "RESET"
            OnMouseClick: toggle Velocity.RES_BUTTON
        Lamp1 (62,115 70x70), variable: Velocity.errorDiode, style: Lamp-Lamp1-Yellow
        Label (70,5 288x97), "Error caused by external force"
END_VISUALIZATION
